PROGRAM MAIN
VAR
	fbModeSelector : FB_ModeSelector;	
END_VAR

fbModeSelector(bControlBox := TRUE);

END_PROGRAM

(* stored: Version 1.1.0.1, ProductVersion 3.1.4024.12
   POU MAIN: Id {134ce0fc-6d16-44c6-b69e-adf0e685ef00}, SpecialFunc None *)
